FUNCTION_BLOCK SamplesAutomationRunner EXTENDS TOF_AutomationEngine.AutomationRunner<2>
VAR_OUTPUT
	SignalControlledIntersectionAutomationController : SignalControlledIntersectionAutomationController(THIS^);
	
	DemoWorkflowAutomationController : DemoWorkflowAutomationController(THIS^);
END_VAR
VAR
	_ClassName : STRING := __POUNAME();
	
	_AutomationControllers : ARRAY [0..1] OF TOF_AutomationEngine.IAutomationController := 
	[
		SignalControlledIntersectionAutomationController,
		DemoWorkflowAutomationController
	];
END_VAR

{attribute 'monitoring' := 'call'}
PROPERTY ClassName : STRING
GET
ClassName := _ClassName;
END_GET
END_PROPERTY

{attribute 'monitoring' := 'call'}
PROPERTY Controllers : REFERENCE TO ARRAY [0.._ControllerCount - 1] OF TOF_AutomationEngine.IAutomationController
GET
Controllers REF= _AutomationControllers;
END_GET
END_PROPERTY

//FB_Init is always available implicitly and it is used primarily for initialization.
//The return value is not evaluated. For a specific influence, you can also declare the
//methods explicitly and provide additional code there with the standard initialization
//code. You can evaluate the return value.
METHOD FB_Init: BOOL
VAR_INPUT
    bInitRetains: BOOL; // TRUE: the retain variables are initialized (reset warm / reset cold)
    bInCopyCode: BOOL;  // TRUE: the instance will be copied to the copy code afterward (online change)   
END_VAR
SignalControlledIntersectionAutomationController.SetSimulationMode(TRUE);
DemoWorkflowAutomationController.SetSimulationMode(TRUE);
END_METHOD

{attribute 'monitoring' := 'call'}
PROPERTY NamespaceName : STRING
GET
NamespaceName := CurrentNamespace.Name;
END_GET
END_PROPERTY

{attribute 'monitoring' := 'call'}
PROPERTY SelfSize : ULINT
GET
SelfSize := XSIZEOF(THIS^);
END_GET
END_PROPERTY

END_FUNCTION_BLOCK

(* stored: Version 1.1.0.1
   POU SamplesAutomationRunner: Id {ff964406-6e7d-46be-9bc3-ae0ec1a8df3e}, SpecialFunc None
   Property ClassName: Id {44015b9d-a297-4fcc-8765-1882288ab888}
   Get Get: Id {cab8ddbf-0d31-4c51-ad36-9a0a06b1f991}
   Property Controllers: Id {6362bba8-7b43-445e-977a-8defd358fba7}
   Get Get: Id {fccbb52a-40a3-46d6-904d-074ece3ee424}
   Method FB_Init: Id {9c8ff6ec-3304-47ad-8fa3-9fc9a9937959}
   Property NamespaceName: Id {1188c0db-1edb-4fa4-8493-18f524ca89e4}
   Get Get: Id {120fe509-6026-468f-b248-0ce4722cb6be}
   Property SelfSize: Id {23eac530-e293-442f-b701-6a55d41e89b4}
   Get Get: Id {6b2e6577-47f6-43bc-b255-c7867b3833f7} *)
